// TIA Portal V16 export
// export: Created 2026-06-22T07:42:12.2698946Z, ExportSetting WithDefaults, DisplayName Totally Integrated Automation Portal, DisplayVersion V16 Update 8, DisplayName TIA Portal Version Control Interface, DisplayVersion V16 Update 8, DisplayName TIA Portal Openness, DisplayVersion V16 Update 8, DisplayName SINAMICS Startdrive Advanced, DisplayVersion V16, DisplayName SINAMICS Startdrive G130, G150, S120, S150, SINAMICS MV, S210, DisplayVersion V16, DisplayName SINAMICS Startdrive G110M, G120, G120C, G120D, G120P, DisplayVersion V16, DisplayName STEP 7 Professional, DisplayVersion V16 Update 8, DisplayName STEP 7 Safety, DisplayVersion V16 Update 7, DisplayName WinCC Advanced, DisplayVersion V16 Update 8
TagTable "默认变量表"
  Button : Bool  (1 s)
  Light : Bool  (1 s)
  IOField : Int  (1 s)
  IOField_1 : Int  (1 s)
  IO_Elevator_Floor : Int  (1 s)
  STS_Elevator_Running : Bool  (1 s)
  STS_Elevator_Up : Bool  (1 s)
  STS_Elevator_Down : Bool  (1 s)
  STS_Elevator_DoorOpen : Bool  (1 s)
  LMP_Elevator_Fault : Bool  (1 s)
  BTN_Elevator_Up : Bool  (1 s)
  BTN_Elevator_Down : Bool  (1 s)
  MEM_Elevator_EmergencyStop : Bool  (1 s)
